// TIA Portal V16 export
// export: Created 2023-03-29T11:03:26.8705636Z, ExportSetting WithDefaults, DisplayName Totally Integrated Automation Portal, DisplayVersion V16 Update 6, DisplayName TIA Portal Version Control Interface, DisplayVersion V16 Update 2, DisplayName TIA Portal Openness, DisplayVersion V16 Update 6, DisplayName STEP 7 Professional, DisplayVersion V16 Update 6, DisplayName STEP 7 Safety, DisplayVersion V16, DisplayName WinCC Advanced, DisplayVersion V16 Update 6
FUNCTION "Read_MPP04_2_ModbusRTU" : Void   // FC24, LAD
TITLE = Odczyt parametrów z MPP04 Pompownia / Read data from SC100
{ S7_Optimized_Access := 'TRUE' }
AUTHOR : rtecmer
VERSION : 0.1
// Czytanie z przepływomierza pompownia główna. Modbus RTU 19200, bit stop-1, parti-no
// Czytanie z SC1000 
// Obsługa protokołu Master Modbus RTU.  Odczyt pomiarów  i status czujnika SC1000
// stored: AutoNumber false, IsIECCheckEnabled false, SetENOAutomatically false, UDAEnableTagReadback false
   VAR_TEMP
      Wielkość_przeływu_Adres0_0 : DWord;
      Wielkość_przeływu_Adres0_1 : DWord;
      Wielkość_przeływu_Adres2_0 : DWord;
      Wielkość_przeływu_Adres2_2 : DWord;
   END_VAR
   VAR_TEMP   // added for the SCL form of the ladder/FBD networks
      _w1 : Bool;
      _w2 : Bool;
   END_VAR
BEGIN

REGION Network 1: Odczyt parametrów z MPP04 Studnia na tłocznym
   // Czytanie z przepływomierza pompownia główna. Modbus RTU 19200, bit stop-1, parti-no
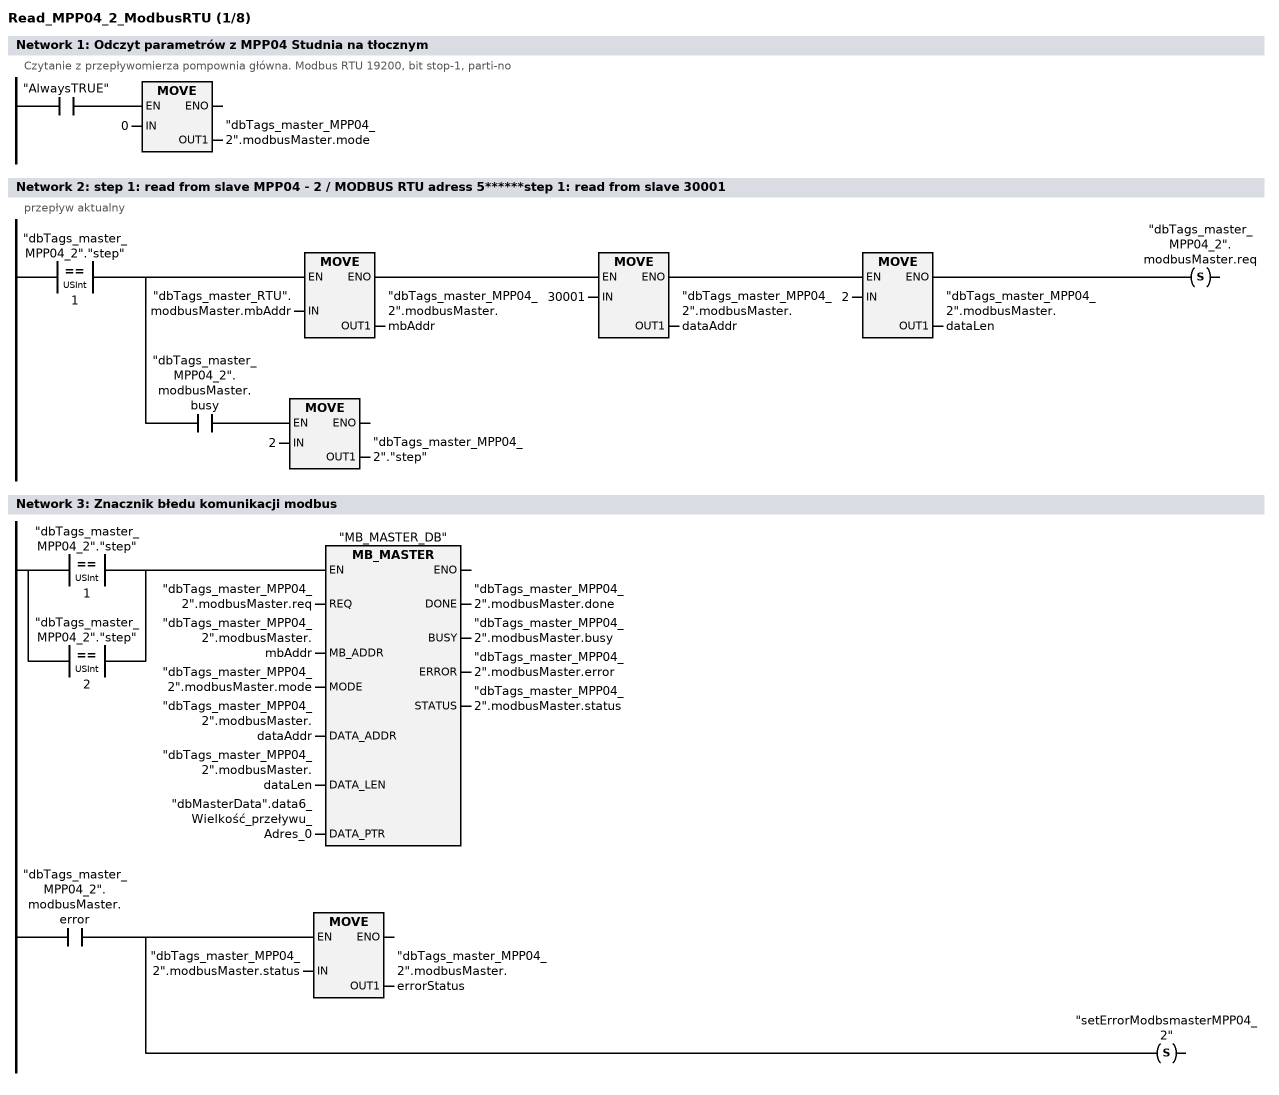
   RUNG wire#powerrail
      Contact( "AlwaysTRUE" )
      { S7_GenerateENO := "TRUE" } Move(in := 0, out1 => "dbTags_master_MPP04_2".modbusMaster.mode)
   END_RUNG
   // the same network as SCL:
   IF "AlwaysTRUE" THEN "dbTags_master_MPP04_2".modbusMaster.mode := 0; END_IF;
END_REGION

REGION Network 2: step 1: read from slave MPP04 - 2 / MODBUS RTU adress 5******step 1: read from slave 30001
   // przepływ aktualny
   RUNG wire#powerrail
      { S7_Templates := "SrcType := USInt" } EQ_Contact(in1 := "dbTags_master_MPP04_2"."step", in2 := 1)
      wire#w1
      Move(in := "dbTags_master_RTU".modbusMaster.mbAddr, out1 => "dbTags_master_MPP04_2".modbusMaster.mbAddr)
      { S7_GenerateENO := "TRUE" } Move(in := 30001, out1 => "dbTags_master_MPP04_2".modbusMaster.dataAddr)
      Move(in := 2, out1 => "dbTags_master_MPP04_2".modbusMaster.dataLen)
      S_Coil( "dbTags_master_MPP04_2".modbusMaster.req )
   END_RUNG
   RUNG wire#w1
      Contact( "dbTags_master_MPP04_2".modbusMaster.busy )
      { S7_GenerateENO := "TRUE" } Move(in := 2, out1 => "dbTags_master_MPP04_2"."step")
   END_RUNG
   // the same network as SCL:
   // ENO of a box is taken as its EN; it also drops when the box reports an error
   #_w1 := "dbTags_master_MPP04_2"."step" = 1;
   IF #_w1 THEN
       "dbTags_master_MPP04_2".modbusMaster.mbAddr := "dbTags_master_RTU".modbusMaster.mbAddr;
       "dbTags_master_MPP04_2".modbusMaster.dataAddr := 30001;
       "dbTags_master_MPP04_2".modbusMaster.dataLen := 2;
       "dbTags_master_MPP04_2".modbusMaster.req := TRUE;
   END_IF;
   IF #_w1 AND "dbTags_master_MPP04_2".modbusMaster.busy THEN "dbTags_master_MPP04_2"."step" := 2; END_IF;
END_REGION

REGION Network 3: Znacznik błedu komunikacji modbus
   RUNG wire#powerrail
      { S7_Templates := "SrcType := USInt" } EQ_Contact(in1 := "dbTags_master_MPP04_2"."step", in2 := 1)
      wire#w1
      "MB_MASTER_DB".MB_MASTER(REQ := "dbTags_master_MPP04_2".modbusMaster.req, MB_ADDR := "dbTags_master_MPP04_2".modbusMaster.mbAddr, MODE := "dbTags_master_MPP04_2".modbusMaster.mode, DATA_ADDR := "dbTags_master_MPP04_2".modbusMaster.dataAddr, DATA_LEN := "dbTags_master_MPP04_2".modbusMaster.dataLen, DATA_PTR := "dbMasterData".data6_Wielkość_przeływu_Adres_0, DONE => "dbTags_master_MPP04_2".modbusMaster.done, BUSY => "dbTags_master_MPP04_2".modbusMaster.busy, ERROR => "dbTags_master_MPP04_2".modbusMaster.error, STATUS => "dbTags_master_MPP04_2".modbusMaster.status)
   END_RUNG
   RUNG wire#powerrail
      { S7_Templates := "SrcType := USInt" } EQ_Contact(in1 := "dbTags_master_MPP04_2"."step", in2 := 2)
   END_RUNG wire#w1
   RUNG wire#powerrail
      Contact( "dbTags_master_MPP04_2".modbusMaster.error )
      wire#w2
      { S7_GenerateENO := "TRUE" } Move(in := "dbTags_master_MPP04_2".modbusMaster.status, out1 => "dbTags_master_MPP04_2".modbusMaster.errorStatus)
   END_RUNG
   RUNG wire#w2
      S_Coil( "setErrorModbsmasterMPP04_2" )
   END_RUNG
   // the same network as SCL:
   IF ("dbTags_master_MPP04_2"."step" = 1) OR ("dbTags_master_MPP04_2"."step" = 2) THEN
       "MB_MASTER_DB"(REQ := "dbTags_master_MPP04_2".modbusMaster.req,   // MB_MASTER
                      MB_ADDR := "dbTags_master_MPP04_2".modbusMaster.mbAddr,
                      MODE := "dbTags_master_MPP04_2".modbusMaster.mode,
                      DATA_ADDR := "dbTags_master_MPP04_2".modbusMaster.dataAddr,
                      DATA_LEN := "dbTags_master_MPP04_2".modbusMaster.dataLen,
                      DATA_PTR := "dbMasterData".data6_Wielkość_przeływu_Adres_0,
                      DONE => "dbTags_master_MPP04_2".modbusMaster.done,
                      BUSY => "dbTags_master_MPP04_2".modbusMaster.busy,
                      ERROR => "dbTags_master_MPP04_2".modbusMaster.error,
                      STATUS => "dbTags_master_MPP04_2".modbusMaster.status);
   END_IF;
   IF "dbTags_master_MPP04_2".modbusMaster.error THEN
       "dbTags_master_MPP04_2".modbusMaster.errorStatus := "dbTags_master_MPP04_2".modbusMaster.status;
       "setErrorModbsmasterMPP04_2" := TRUE;
   END_IF;
END_REGION

REGION Network 4: step 4: save received data / step 2: save received data 30001
   // Pomiar Temperatury KDN1
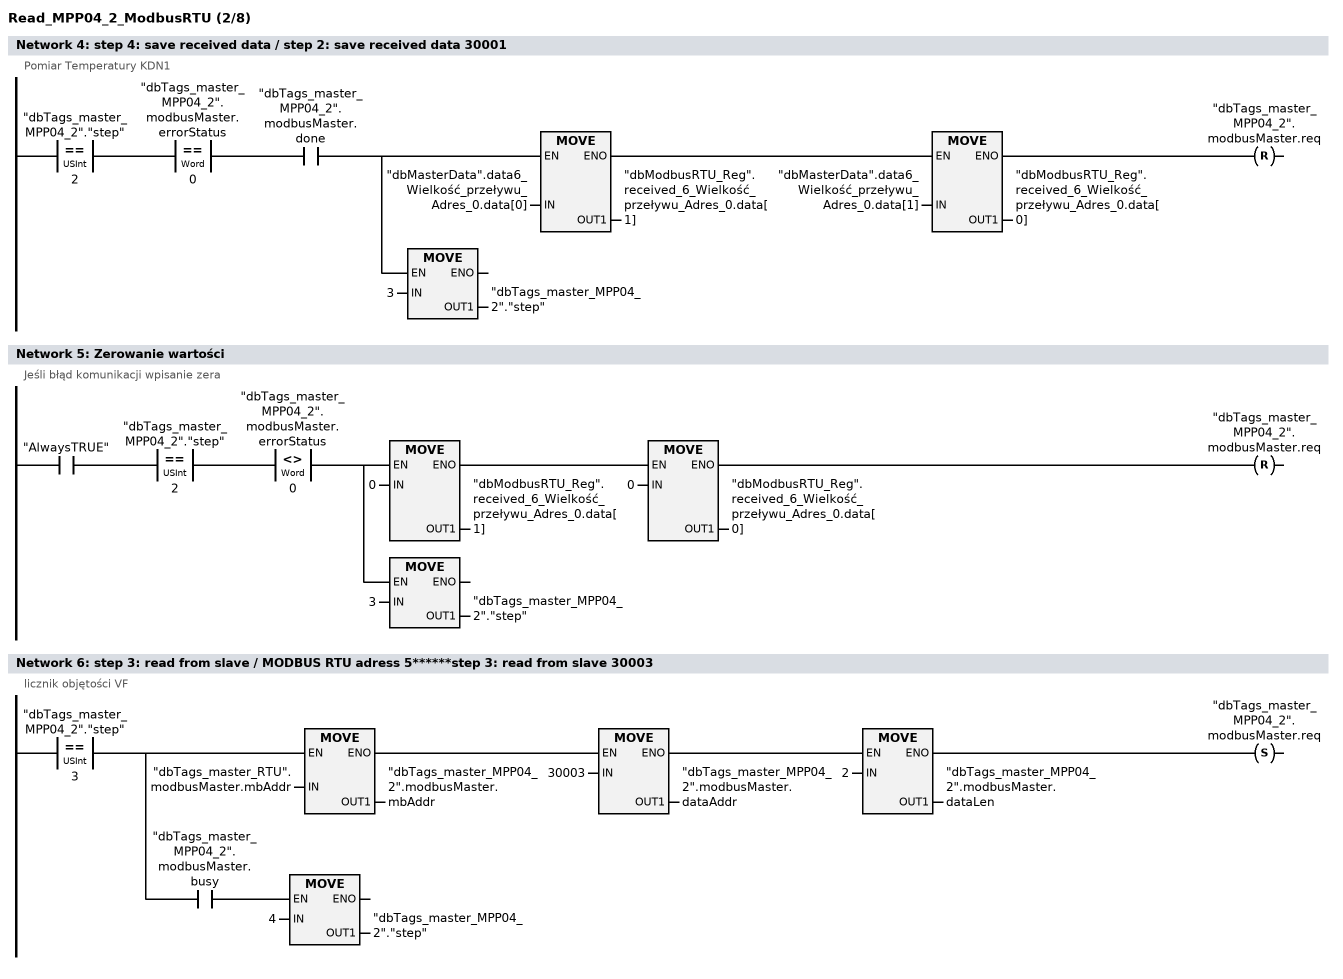
   RUNG wire#powerrail
      { S7_Templates := "SrcType := USInt" } EQ_Contact(in1 := "dbTags_master_MPP04_2"."step", in2 := 2)
      { S7_Templates := "SrcType := Word" } EQ_Contact(in1 := "dbTags_master_MPP04_2".modbusMaster.errorStatus, in2 := 0)
      Contact( "dbTags_master_MPP04_2".modbusMaster.done )
      wire#w1
      { S7_GenerateENO := "TRUE" } Move(in := "dbMasterData".data6_Wielkość_przeływu_Adres_0.data[0], out1 => "dbModbusRTU_Reg".received_6_Wielkość_przeływu_Adres_0.data[1])
      { S7_GenerateENO := "TRUE" } Move(in := "dbMasterData".data6_Wielkość_przeływu_Adres_0.data[1], out1 => "dbModbusRTU_Reg".received_6_Wielkość_przeływu_Adres_0.data[0])
      R_Coil( "dbTags_master_MPP04_2".modbusMaster.req )
   END_RUNG
   RUNG wire#w1
      { S7_GenerateENO := "TRUE" } Move(in := 3, out1 => "dbTags_master_MPP04_2"."step")
   END_RUNG
   // the same network as SCL:
   // ENO of a box is taken as its EN; it also drops when the box reports an error
   IF ("dbTags_master_MPP04_2"."step" = 2) AND ("dbTags_master_MPP04_2".modbusMaster.errorStatus = 0) AND "dbTags_master_MPP04_2".modbusMaster.done THEN
       "dbModbusRTU_Reg".received_6_Wielkość_przeływu_Adres_0.data[1] := "dbMasterData".data6_Wielkość_przeływu_Adres_0.data[0];
       "dbModbusRTU_Reg".received_6_Wielkość_przeływu_Adres_0.data[0] := "dbMasterData".data6_Wielkość_przeływu_Adres_0.data[1];
       "dbTags_master_MPP04_2".modbusMaster.req := FALSE;
       "dbTags_master_MPP04_2"."step" := 3;
   END_IF;
END_REGION

REGION Network 5: Zerowanie wartości
   // Jeśli błąd komunikacji wpisanie zera
   RUNG wire#powerrail
      Contact( "AlwaysTRUE" )
      { S7_Templates := "SrcType := USInt" } EQ_Contact(in1 := "dbTags_master_MPP04_2"."step", in2 := 2)
      { S7_Templates := "SrcType := Word" } NE_Contact(in1 := "dbTags_master_MPP04_2".modbusMaster.errorStatus, in2 := 0)
      wire#w1
      { S7_GenerateENO := "TRUE" } Move(in := 0, out1 => "dbModbusRTU_Reg".received_6_Wielkość_przeływu_Adres_0.data[1])
      { S7_GenerateENO := "TRUE" } Move(in := 0, out1 => "dbModbusRTU_Reg".received_6_Wielkość_przeływu_Adres_0.data[0])
      R_Coil( "dbTags_master_MPP04_2".modbusMaster.req )
   END_RUNG
   RUNG wire#w1
      { S7_GenerateENO := "TRUE" } Move(in := 3, out1 => "dbTags_master_MPP04_2"."step")
   END_RUNG
   // the same network as SCL:
   // ENO of a box is taken as its EN; it also drops when the box reports an error
   IF "AlwaysTRUE" AND ("dbTags_master_MPP04_2"."step" = 2) AND ("dbTags_master_MPP04_2".modbusMaster.errorStatus <> 0) THEN
       "dbModbusRTU_Reg".received_6_Wielkość_przeływu_Adres_0.data[1] := 0;
       "dbModbusRTU_Reg".received_6_Wielkość_przeływu_Adres_0.data[0] := 0;
       "dbTags_master_MPP04_2".modbusMaster.req := FALSE;
       "dbTags_master_MPP04_2"."step" := 3;
   END_IF;
END_REGION

REGION Network 6: step 3: read from slave / MODBUS RTU adress 5******step 3: read from slave 30003
   // licznik objętości VF
   RUNG wire#powerrail
      { S7_Templates := "SrcType := USInt" } EQ_Contact(in1 := "dbTags_master_MPP04_2"."step", in2 := 3)
      wire#w1
      Move(in := "dbTags_master_RTU".modbusMaster.mbAddr, out1 => "dbTags_master_MPP04_2".modbusMaster.mbAddr)
      { S7_GenerateENO := "TRUE" } Move(in := 30003, out1 => "dbTags_master_MPP04_2".modbusMaster.dataAddr)
      Move(in := 2, out1 => "dbTags_master_MPP04_2".modbusMaster.dataLen)
      S_Coil( "dbTags_master_MPP04_2".modbusMaster.req )
   END_RUNG
   RUNG wire#w1
      Contact( "dbTags_master_MPP04_2".modbusMaster.busy )
      { S7_GenerateENO := "TRUE" } Move(in := 4, out1 => "dbTags_master_MPP04_2"."step")
   END_RUNG
   // the same network as SCL:
   // ENO of a box is taken as its EN; it also drops when the box reports an error
   #_w1 := "dbTags_master_MPP04_2"."step" = 3;
   IF #_w1 THEN
       "dbTags_master_MPP04_2".modbusMaster.mbAddr := "dbTags_master_RTU".modbusMaster.mbAddr;
       "dbTags_master_MPP04_2".modbusMaster.dataAddr := 30003;
       "dbTags_master_MPP04_2".modbusMaster.dataLen := 2;
       "dbTags_master_MPP04_2".modbusMaster.req := TRUE;
   END_IF;
   IF #_w1 AND "dbTags_master_MPP04_2".modbusMaster.busy THEN "dbTags_master_MPP04_2"."step" := 4; END_IF;
END_REGION

REGION Network 7: Znacznik błedu komunikacji modbus
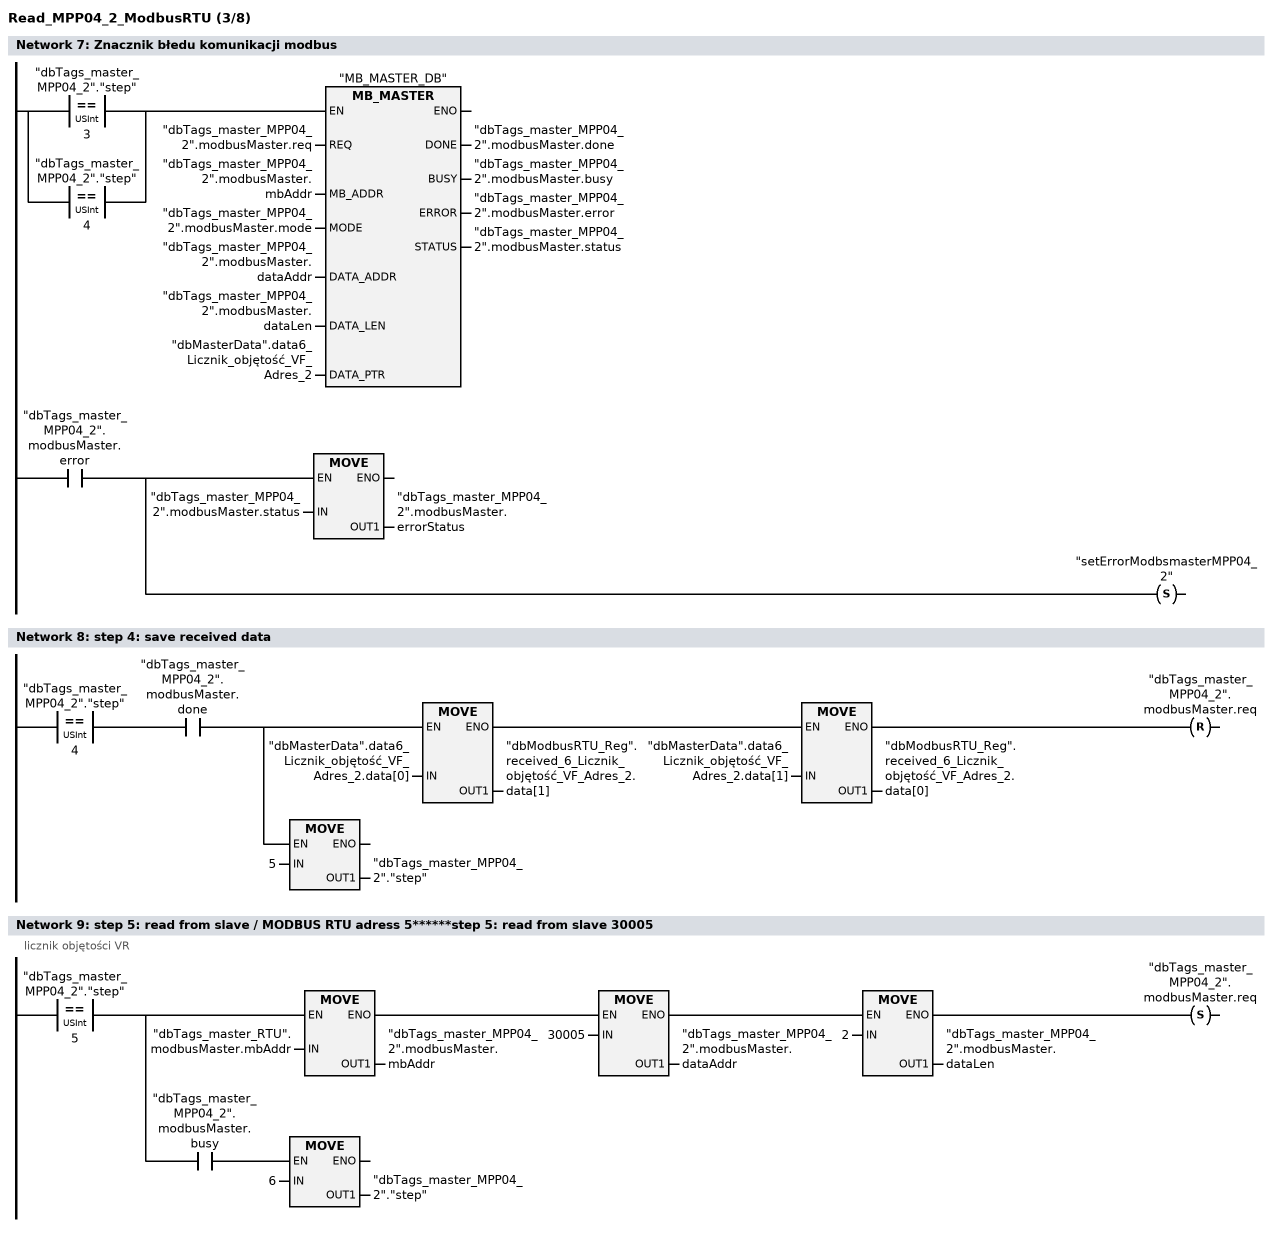
   RUNG wire#powerrail
      { S7_Templates := "SrcType := USInt" } EQ_Contact(in1 := "dbTags_master_MPP04_2"."step", in2 := 3)
      wire#w1
      "MB_MASTER_DB".MB_MASTER(REQ := "dbTags_master_MPP04_2".modbusMaster.req, MB_ADDR := "dbTags_master_MPP04_2".modbusMaster.mbAddr, MODE := "dbTags_master_MPP04_2".modbusMaster.mode, DATA_ADDR := "dbTags_master_MPP04_2".modbusMaster.dataAddr, DATA_LEN := "dbTags_master_MPP04_2".modbusMaster.dataLen, DATA_PTR := "dbMasterData".data6_Licznik_objętość_VF_Adres_2, DONE => "dbTags_master_MPP04_2".modbusMaster.done, BUSY => "dbTags_master_MPP04_2".modbusMaster.busy, ERROR => "dbTags_master_MPP04_2".modbusMaster.error, STATUS => "dbTags_master_MPP04_2".modbusMaster.status)
   END_RUNG
   RUNG wire#powerrail
      { S7_Templates := "SrcType := USInt" } EQ_Contact(in1 := "dbTags_master_MPP04_2"."step", in2 := 4)
   END_RUNG wire#w1
   RUNG wire#powerrail
      Contact( "dbTags_master_MPP04_2".modbusMaster.error )
      wire#w2
      { S7_GenerateENO := "TRUE" } Move(in := "dbTags_master_MPP04_2".modbusMaster.status, out1 => "dbTags_master_MPP04_2".modbusMaster.errorStatus)
   END_RUNG
   RUNG wire#w2
      S_Coil( "setErrorModbsmasterMPP04_2" )
   END_RUNG
   // the same network as SCL:
   IF ("dbTags_master_MPP04_2"."step" = 3) OR ("dbTags_master_MPP04_2"."step" = 4) THEN
       "MB_MASTER_DB"(REQ := "dbTags_master_MPP04_2".modbusMaster.req,   // MB_MASTER
                      MB_ADDR := "dbTags_master_MPP04_2".modbusMaster.mbAddr,
                      MODE := "dbTags_master_MPP04_2".modbusMaster.mode,
                      DATA_ADDR := "dbTags_master_MPP04_2".modbusMaster.dataAddr,
                      DATA_LEN := "dbTags_master_MPP04_2".modbusMaster.dataLen,
                      DATA_PTR := "dbMasterData".data6_Licznik_objętość_VF_Adres_2,
                      DONE => "dbTags_master_MPP04_2".modbusMaster.done,
                      BUSY => "dbTags_master_MPP04_2".modbusMaster.busy,
                      ERROR => "dbTags_master_MPP04_2".modbusMaster.error,
                      STATUS => "dbTags_master_MPP04_2".modbusMaster.status);
   END_IF;
   IF "dbTags_master_MPP04_2".modbusMaster.error THEN
       "dbTags_master_MPP04_2".modbusMaster.errorStatus := "dbTags_master_MPP04_2".modbusMaster.status;
       "setErrorModbsmasterMPP04_2" := TRUE;
   END_IF;
END_REGION

REGION Network 8: step 4: save received data
   RUNG wire#powerrail
      { S7_Templates := "SrcType := USInt" } EQ_Contact(in1 := "dbTags_master_MPP04_2"."step", in2 := 4)
      Contact( "dbTags_master_MPP04_2".modbusMaster.done )
      wire#w1
      { S7_GenerateENO := "TRUE" } Move(in := "dbMasterData".data6_Licznik_objętość_VF_Adres_2.data[0], out1 => "dbModbusRTU_Reg".received_6_Licznik_objętość_VF_Adres_2.data[1])
      { S7_GenerateENO := "TRUE" } Move(in := "dbMasterData".data6_Licznik_objętość_VF_Adres_2.data[1], out1 => "dbModbusRTU_Reg".received_6_Licznik_objętość_VF_Adres_2.data[0])
      R_Coil( "dbTags_master_MPP04_2".modbusMaster.req )
   END_RUNG
   RUNG wire#w1
      { S7_GenerateENO := "TRUE" } Move(in := 5, out1 => "dbTags_master_MPP04_2"."step")
   END_RUNG
   // the same network as SCL:
   // ENO of a box is taken as its EN; it also drops when the box reports an error
   IF ("dbTags_master_MPP04_2"."step" = 4) AND "dbTags_master_MPP04_2".modbusMaster.done THEN
       "dbModbusRTU_Reg".received_6_Licznik_objętość_VF_Adres_2.data[1] := "dbMasterData".data6_Licznik_objętość_VF_Adres_2.data[0];
       "dbModbusRTU_Reg".received_6_Licznik_objętość_VF_Adres_2.data[0] := "dbMasterData".data6_Licznik_objętość_VF_Adres_2.data[1];
       "dbTags_master_MPP04_2".modbusMaster.req := FALSE;
       "dbTags_master_MPP04_2"."step" := 5;
   END_IF;
END_REGION

REGION Network 9: step 5: read from slave / MODBUS RTU adress 5******step 5: read from slave 30005
   // licznik objętości VR
   RUNG wire#powerrail
      { S7_Templates := "SrcType := USInt" } EQ_Contact(in1 := "dbTags_master_MPP04_2"."step", in2 := 5)
      wire#w1
      Move(in := "dbTags_master_RTU".modbusMaster.mbAddr, out1 => "dbTags_master_MPP04_2".modbusMaster.mbAddr)
      { S7_GenerateENO := "TRUE" } Move(in := 30005, out1 => "dbTags_master_MPP04_2".modbusMaster.dataAddr)
      Move(in := 2, out1 => "dbTags_master_MPP04_2".modbusMaster.dataLen)
      S_Coil( "dbTags_master_MPP04_2".modbusMaster.req )
   END_RUNG
   RUNG wire#w1
      Contact( "dbTags_master_MPP04_2".modbusMaster.busy )
      { S7_GenerateENO := "TRUE" } Move(in := 6, out1 => "dbTags_master_MPP04_2"."step")
   END_RUNG
   // the same network as SCL:
   // ENO of a box is taken as its EN; it also drops when the box reports an error
   #_w1 := "dbTags_master_MPP04_2"."step" = 5;
   IF #_w1 THEN
       "dbTags_master_MPP04_2".modbusMaster.mbAddr := "dbTags_master_RTU".modbusMaster.mbAddr;
       "dbTags_master_MPP04_2".modbusMaster.dataAddr := 30005;
       "dbTags_master_MPP04_2".modbusMaster.dataLen := 2;
       "dbTags_master_MPP04_2".modbusMaster.req := TRUE;
   END_IF;
   IF #_w1 AND "dbTags_master_MPP04_2".modbusMaster.busy THEN "dbTags_master_MPP04_2"."step" := 6; END_IF;
END_REGION

REGION Network 10: Znacznik błedu komunikacji modbus
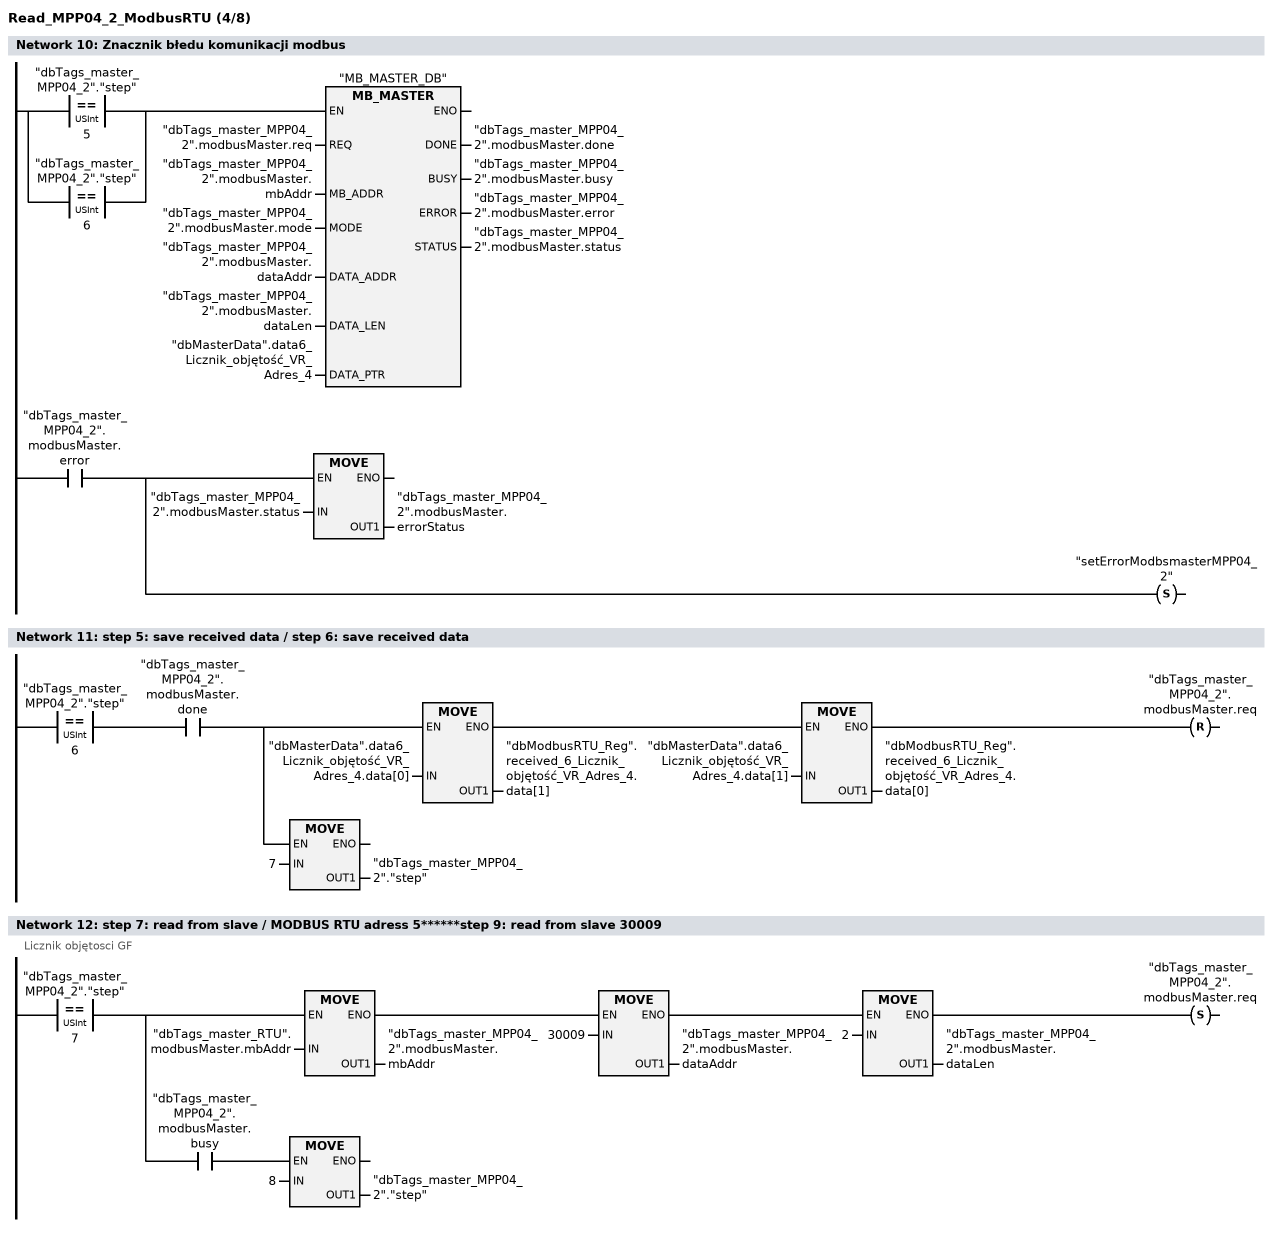
   RUNG wire#powerrail
      { S7_Templates := "SrcType := USInt" } EQ_Contact(in1 := "dbTags_master_MPP04_2"."step", in2 := 5)
      wire#w1
      "MB_MASTER_DB".MB_MASTER(REQ := "dbTags_master_MPP04_2".modbusMaster.req, MB_ADDR := "dbTags_master_MPP04_2".modbusMaster.mbAddr, MODE := "dbTags_master_MPP04_2".modbusMaster.mode, DATA_ADDR := "dbTags_master_MPP04_2".modbusMaster.dataAddr, DATA_LEN := "dbTags_master_MPP04_2".modbusMaster.dataLen, DATA_PTR := "dbMasterData".data6_Licznik_objętość_VR_Adres_4, DONE => "dbTags_master_MPP04_2".modbusMaster.done, BUSY => "dbTags_master_MPP04_2".modbusMaster.busy, ERROR => "dbTags_master_MPP04_2".modbusMaster.error, STATUS => "dbTags_master_MPP04_2".modbusMaster.status)
   END_RUNG
   RUNG wire#powerrail
      { S7_Templates := "SrcType := USInt" } EQ_Contact(in1 := "dbTags_master_MPP04_2"."step", in2 := 6)
   END_RUNG wire#w1
   RUNG wire#powerrail
      Contact( "dbTags_master_MPP04_2".modbusMaster.error )
      wire#w2
      { S7_GenerateENO := "TRUE" } Move(in := "dbTags_master_MPP04_2".modbusMaster.status, out1 => "dbTags_master_MPP04_2".modbusMaster.errorStatus)
   END_RUNG
   RUNG wire#w2
      S_Coil( "setErrorModbsmasterMPP04_2" )
   END_RUNG
   // the same network as SCL:
   IF ("dbTags_master_MPP04_2"."step" = 5) OR ("dbTags_master_MPP04_2"."step" = 6) THEN
       "MB_MASTER_DB"(REQ := "dbTags_master_MPP04_2".modbusMaster.req,   // MB_MASTER
                      MB_ADDR := "dbTags_master_MPP04_2".modbusMaster.mbAddr,
                      MODE := "dbTags_master_MPP04_2".modbusMaster.mode,
                      DATA_ADDR := "dbTags_master_MPP04_2".modbusMaster.dataAddr,
                      DATA_LEN := "dbTags_master_MPP04_2".modbusMaster.dataLen,
                      DATA_PTR := "dbMasterData".data6_Licznik_objętość_VR_Adres_4,
                      DONE => "dbTags_master_MPP04_2".modbusMaster.done,
                      BUSY => "dbTags_master_MPP04_2".modbusMaster.busy,
                      ERROR => "dbTags_master_MPP04_2".modbusMaster.error,
                      STATUS => "dbTags_master_MPP04_2".modbusMaster.status);
   END_IF;
   IF "dbTags_master_MPP04_2".modbusMaster.error THEN
       "dbTags_master_MPP04_2".modbusMaster.errorStatus := "dbTags_master_MPP04_2".modbusMaster.status;
       "setErrorModbsmasterMPP04_2" := TRUE;
   END_IF;
END_REGION

REGION Network 11: step 5: save received data / step 6: save received data
   RUNG wire#powerrail
      { S7_Templates := "SrcType := USInt" } EQ_Contact(in1 := "dbTags_master_MPP04_2"."step", in2 := 6)
      Contact( "dbTags_master_MPP04_2".modbusMaster.done )
      wire#w1
      { S7_GenerateENO := "TRUE" } Move(in := "dbMasterData".data6_Licznik_objętość_VR_Adres_4.data[0], out1 => "dbModbusRTU_Reg".received_6_Licznik_objętość_VR_Adres_4.data[1])
      { S7_GenerateENO := "TRUE" } Move(in := "dbMasterData".data6_Licznik_objętość_VR_Adres_4.data[1], out1 => "dbModbusRTU_Reg".received_6_Licznik_objętość_VR_Adres_4.data[0])
      R_Coil( "dbTags_master_MPP04_2".modbusMaster.req )
   END_RUNG
   RUNG wire#w1
      { S7_GenerateENO := "TRUE" } Move(in := 7, out1 => "dbTags_master_MPP04_2"."step")
   END_RUNG
   // the same network as SCL:
   // ENO of a box is taken as its EN; it also drops when the box reports an error
   IF ("dbTags_master_MPP04_2"."step" = 6) AND "dbTags_master_MPP04_2".modbusMaster.done THEN
       "dbModbusRTU_Reg".received_6_Licznik_objętość_VR_Adres_4.data[1] := "dbMasterData".data6_Licznik_objętość_VR_Adres_4.data[0];
       "dbModbusRTU_Reg".received_6_Licznik_objętość_VR_Adres_4.data[0] := "dbMasterData".data6_Licznik_objętość_VR_Adres_4.data[1];
       "dbTags_master_MPP04_2".modbusMaster.req := FALSE;
       "dbTags_master_MPP04_2"."step" := 7;
   END_IF;
END_REGION

REGION Network 12: step 7: read from slave / MODBUS RTU adress 5******step 9: read from slave 30009
   // Licznik objętosci GF
   RUNG wire#powerrail
      { S7_Templates := "SrcType := USInt" } EQ_Contact(in1 := "dbTags_master_MPP04_2"."step", in2 := 7)
      wire#w1
      Move(in := "dbTags_master_RTU".modbusMaster.mbAddr, out1 => "dbTags_master_MPP04_2".modbusMaster.mbAddr)
      { S7_GenerateENO := "TRUE" } Move(in := 30009, out1 => "dbTags_master_MPP04_2".modbusMaster.dataAddr)
      Move(in := 2, out1 => "dbTags_master_MPP04_2".modbusMaster.dataLen)
      S_Coil( "dbTags_master_MPP04_2".modbusMaster.req )
   END_RUNG
   RUNG wire#w1
      Contact( "dbTags_master_MPP04_2".modbusMaster.busy )
      { S7_GenerateENO := "TRUE" } Move(in := 8, out1 => "dbTags_master_MPP04_2"."step")
   END_RUNG
   // the same network as SCL:
   // ENO of a box is taken as its EN; it also drops when the box reports an error
   #_w1 := "dbTags_master_MPP04_2"."step" = 7;
   IF #_w1 THEN
       "dbTags_master_MPP04_2".modbusMaster.mbAddr := "dbTags_master_RTU".modbusMaster.mbAddr;
       "dbTags_master_MPP04_2".modbusMaster.dataAddr := 30009;
       "dbTags_master_MPP04_2".modbusMaster.dataLen := 2;
       "dbTags_master_MPP04_2".modbusMaster.req := TRUE;
   END_IF;
   IF #_w1 AND "dbTags_master_MPP04_2".modbusMaster.busy THEN "dbTags_master_MPP04_2"."step" := 8; END_IF;
END_REGION

REGION Network 13: Znacznik błedu komunikacji modbus
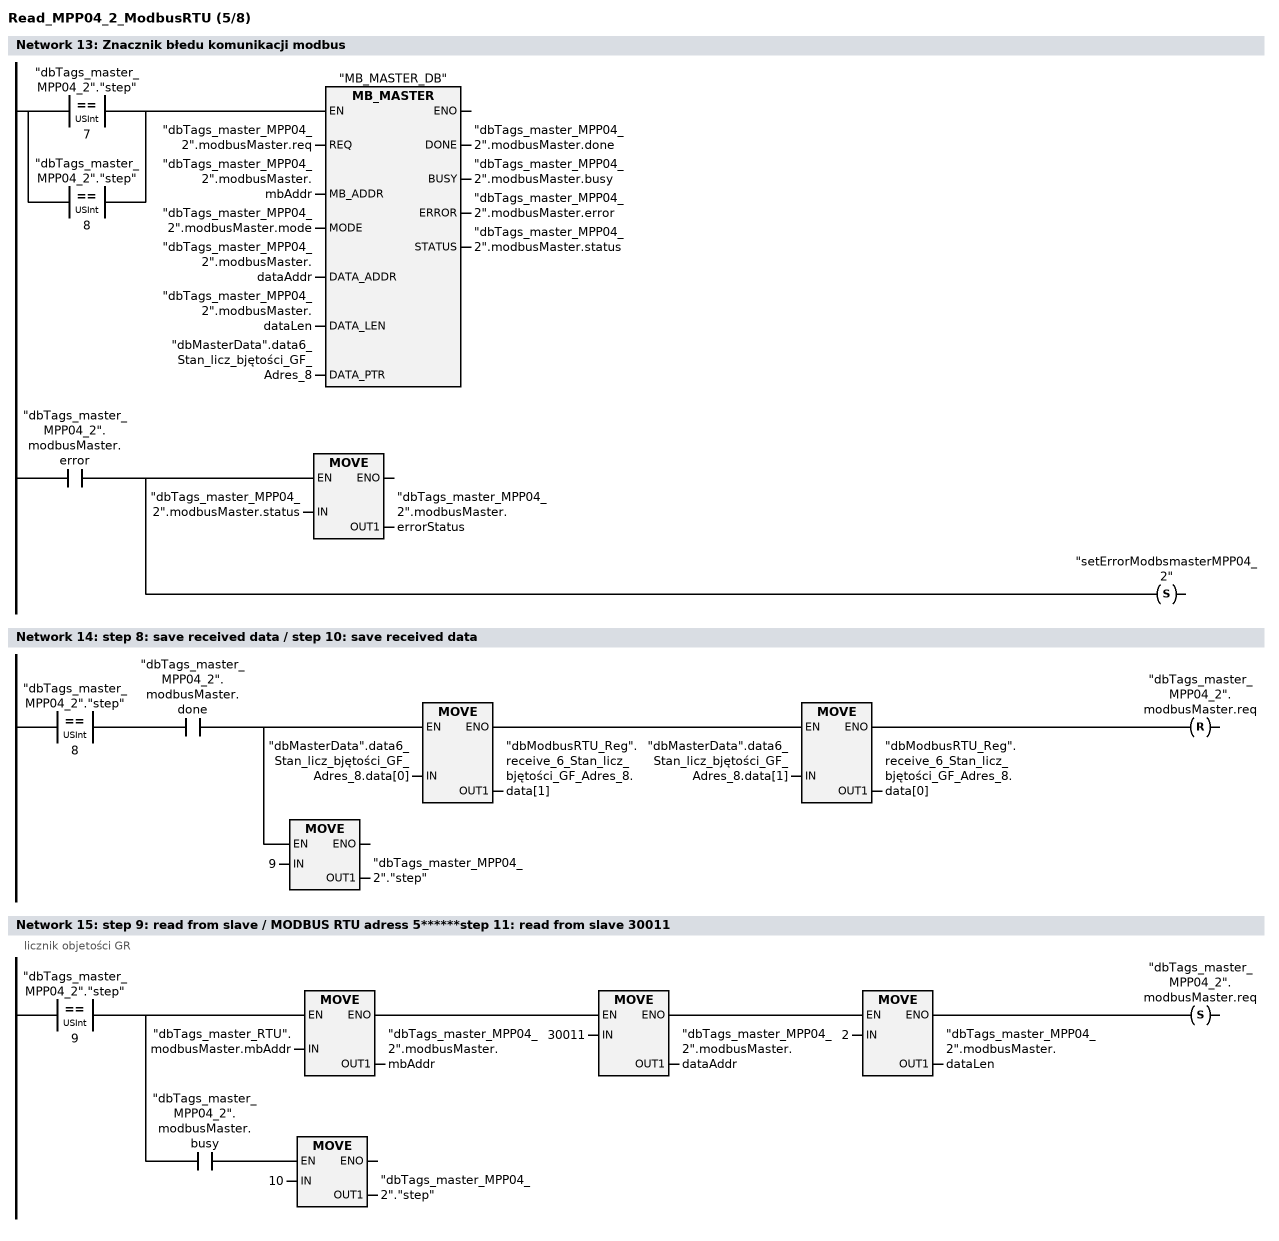
   RUNG wire#powerrail
      { S7_Templates := "SrcType := USInt" } EQ_Contact(in1 := "dbTags_master_MPP04_2"."step", in2 := 7)
      wire#w1
      "MB_MASTER_DB".MB_MASTER(REQ := "dbTags_master_MPP04_2".modbusMaster.req, MB_ADDR := "dbTags_master_MPP04_2".modbusMaster.mbAddr, MODE := "dbTags_master_MPP04_2".modbusMaster.mode, DATA_ADDR := "dbTags_master_MPP04_2".modbusMaster.dataAddr, DATA_LEN := "dbTags_master_MPP04_2".modbusMaster.dataLen, DATA_PTR := "dbMasterData".data6_Stan_licz_bjętości_GF_Adres_8, DONE => "dbTags_master_MPP04_2".modbusMaster.done, BUSY => "dbTags_master_MPP04_2".modbusMaster.busy, ERROR => "dbTags_master_MPP04_2".modbusMaster.error, STATUS => "dbTags_master_MPP04_2".modbusMaster.status)
   END_RUNG
   RUNG wire#powerrail
      { S7_Templates := "SrcType := USInt" } EQ_Contact(in1 := "dbTags_master_MPP04_2"."step", in2 := 8)
   END_RUNG wire#w1
   RUNG wire#powerrail
      Contact( "dbTags_master_MPP04_2".modbusMaster.error )
      wire#w2
      { S7_GenerateENO := "TRUE" } Move(in := "dbTags_master_MPP04_2".modbusMaster.status, out1 => "dbTags_master_MPP04_2".modbusMaster.errorStatus)
   END_RUNG
   RUNG wire#w2
      S_Coil( "setErrorModbsmasterMPP04_2" )
   END_RUNG
   // the same network as SCL:
   IF ("dbTags_master_MPP04_2"."step" = 7) OR ("dbTags_master_MPP04_2"."step" = 8) THEN
       "MB_MASTER_DB"(REQ := "dbTags_master_MPP04_2".modbusMaster.req,   // MB_MASTER
                      MB_ADDR := "dbTags_master_MPP04_2".modbusMaster.mbAddr,
                      MODE := "dbTags_master_MPP04_2".modbusMaster.mode,
                      DATA_ADDR := "dbTags_master_MPP04_2".modbusMaster.dataAddr,
                      DATA_LEN := "dbTags_master_MPP04_2".modbusMaster.dataLen,
                      DATA_PTR := "dbMasterData".data6_Stan_licz_bjętości_GF_Adres_8,
                      DONE => "dbTags_master_MPP04_2".modbusMaster.done,
                      BUSY => "dbTags_master_MPP04_2".modbusMaster.busy,
                      ERROR => "dbTags_master_MPP04_2".modbusMaster.error,
                      STATUS => "dbTags_master_MPP04_2".modbusMaster.status);
   END_IF;
   IF "dbTags_master_MPP04_2".modbusMaster.error THEN
       "dbTags_master_MPP04_2".modbusMaster.errorStatus := "dbTags_master_MPP04_2".modbusMaster.status;
       "setErrorModbsmasterMPP04_2" := TRUE;
   END_IF;
END_REGION

REGION Network 14: step 8: save received data / step 10: save received data
   RUNG wire#powerrail
      { S7_Templates := "SrcType := USInt" } EQ_Contact(in1 := "dbTags_master_MPP04_2"."step", in2 := 8)
      Contact( "dbTags_master_MPP04_2".modbusMaster.done )
      wire#w1
      { S7_GenerateENO := "TRUE" } Move(in := "dbMasterData".data6_Stan_licz_bjętości_GF_Adres_8.data[0], out1 => "dbModbusRTU_Reg".receive_6_Stan_licz_bjętości_GF_Adres_8.data[1])
      { S7_GenerateENO := "TRUE" } Move(in := "dbMasterData".data6_Stan_licz_bjętości_GF_Adres_8.data[1], out1 => "dbModbusRTU_Reg".receive_6_Stan_licz_bjętości_GF_Adres_8.data[0])
      R_Coil( "dbTags_master_MPP04_2".modbusMaster.req )
   END_RUNG
   RUNG wire#w1
      { S7_GenerateENO := "TRUE" } Move(in := 9, out1 => "dbTags_master_MPP04_2"."step")
   END_RUNG
   // the same network as SCL:
   // ENO of a box is taken as its EN; it also drops when the box reports an error
   IF ("dbTags_master_MPP04_2"."step" = 8) AND "dbTags_master_MPP04_2".modbusMaster.done THEN
       "dbModbusRTU_Reg".receive_6_Stan_licz_bjętości_GF_Adres_8.data[1] := "dbMasterData".data6_Stan_licz_bjętości_GF_Adres_8.data[0];
       "dbModbusRTU_Reg".receive_6_Stan_licz_bjętości_GF_Adres_8.data[0] := "dbMasterData".data6_Stan_licz_bjętości_GF_Adres_8.data[1];
       "dbTags_master_MPP04_2".modbusMaster.req := FALSE;
       "dbTags_master_MPP04_2"."step" := 9;
   END_IF;
END_REGION

REGION Network 15: step 9: read from slave / MODBUS RTU adress 5******step 11: read from slave 30011
   // licznik objetości GR
   RUNG wire#powerrail
      { S7_Templates := "SrcType := USInt" } EQ_Contact(in1 := "dbTags_master_MPP04_2"."step", in2 := 9)
      wire#w1
      Move(in := "dbTags_master_RTU".modbusMaster.mbAddr, out1 => "dbTags_master_MPP04_2".modbusMaster.mbAddr)
      { S7_GenerateENO := "TRUE" } Move(in := 30011, out1 => "dbTags_master_MPP04_2".modbusMaster.dataAddr)
      Move(in := 2, out1 => "dbTags_master_MPP04_2".modbusMaster.dataLen)
      S_Coil( "dbTags_master_MPP04_2".modbusMaster.req )
   END_RUNG
   RUNG wire#w1
      Contact( "dbTags_master_MPP04_2".modbusMaster.busy )
      { S7_GenerateENO := "TRUE" } Move(in := 10, out1 => "dbTags_master_MPP04_2"."step")
   END_RUNG
   // the same network as SCL:
   // ENO of a box is taken as its EN; it also drops when the box reports an error
   #_w1 := "dbTags_master_MPP04_2"."step" = 9;
   IF #_w1 THEN
       "dbTags_master_MPP04_2".modbusMaster.mbAddr := "dbTags_master_RTU".modbusMaster.mbAddr;
       "dbTags_master_MPP04_2".modbusMaster.dataAddr := 30011;
       "dbTags_master_MPP04_2".modbusMaster.dataLen := 2;
       "dbTags_master_MPP04_2".modbusMaster.req := TRUE;
   END_IF;
   IF #_w1 AND "dbTags_master_MPP04_2".modbusMaster.busy THEN "dbTags_master_MPP04_2"."step" := 10; END_IF;
END_REGION

REGION Network 16: Znacznik błedu komunikacji modbus
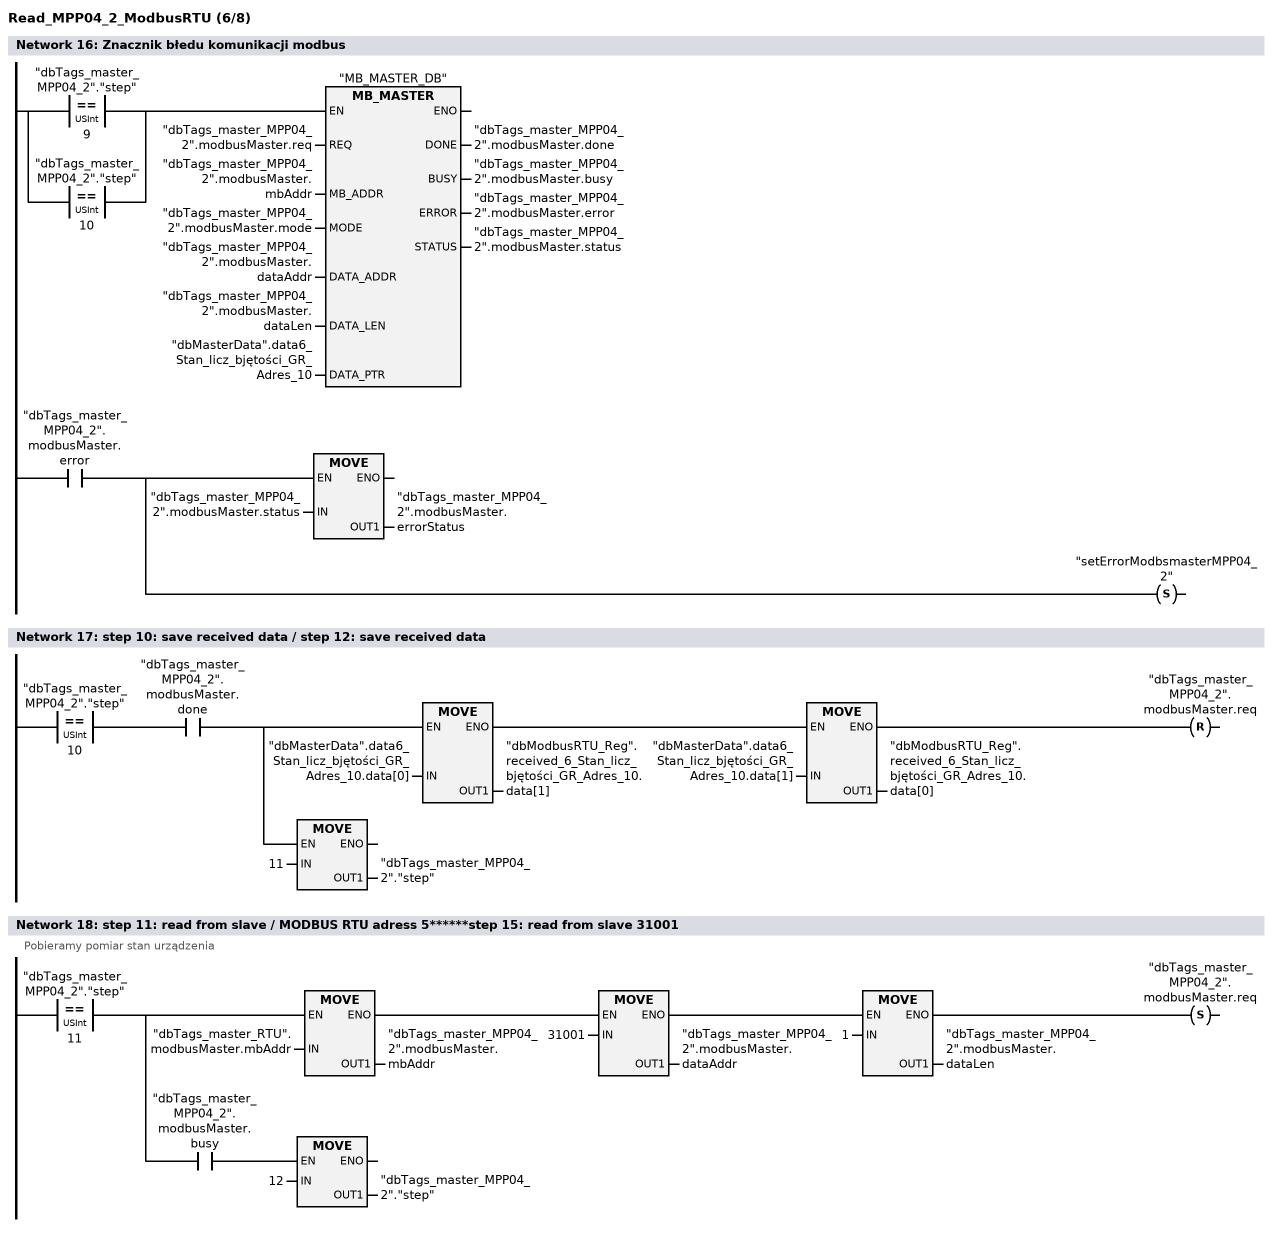
   RUNG wire#powerrail
      { S7_Templates := "SrcType := USInt" } EQ_Contact(in1 := "dbTags_master_MPP04_2"."step", in2 := 9)
      wire#w1
      "MB_MASTER_DB".MB_MASTER(REQ := "dbTags_master_MPP04_2".modbusMaster.req, MB_ADDR := "dbTags_master_MPP04_2".modbusMaster.mbAddr, MODE := "dbTags_master_MPP04_2".modbusMaster.mode, DATA_ADDR := "dbTags_master_MPP04_2".modbusMaster.dataAddr, DATA_LEN := "dbTags_master_MPP04_2".modbusMaster.dataLen, DATA_PTR := "dbMasterData".data6_Stan_licz_bjętości_GR_Adres_10, DONE => "dbTags_master_MPP04_2".modbusMaster.done, BUSY => "dbTags_master_MPP04_2".modbusMaster.busy, ERROR => "dbTags_master_MPP04_2".modbusMaster.error, STATUS => "dbTags_master_MPP04_2".modbusMaster.status)
   END_RUNG
   RUNG wire#powerrail
      { S7_Templates := "SrcType := USInt" } EQ_Contact(in1 := "dbTags_master_MPP04_2"."step", in2 := 10)
   END_RUNG wire#w1
   RUNG wire#powerrail
      Contact( "dbTags_master_MPP04_2".modbusMaster.error )
      wire#w2
      { S7_GenerateENO := "TRUE" } Move(in := "dbTags_master_MPP04_2".modbusMaster.status, out1 => "dbTags_master_MPP04_2".modbusMaster.errorStatus)
   END_RUNG
   RUNG wire#w2
      S_Coil( "setErrorModbsmasterMPP04_2" )
   END_RUNG
   // the same network as SCL:
   IF ("dbTags_master_MPP04_2"."step" = 9) OR ("dbTags_master_MPP04_2"."step" = 10) THEN
       "MB_MASTER_DB"(REQ := "dbTags_master_MPP04_2".modbusMaster.req,   // MB_MASTER
                      MB_ADDR := "dbTags_master_MPP04_2".modbusMaster.mbAddr,
                      MODE := "dbTags_master_MPP04_2".modbusMaster.mode,
                      DATA_ADDR := "dbTags_master_MPP04_2".modbusMaster.dataAddr,
                      DATA_LEN := "dbTags_master_MPP04_2".modbusMaster.dataLen,
                      DATA_PTR := "dbMasterData".data6_Stan_licz_bjętości_GR_Adres_10,
                      DONE => "dbTags_master_MPP04_2".modbusMaster.done,
                      BUSY => "dbTags_master_MPP04_2".modbusMaster.busy,
                      ERROR => "dbTags_master_MPP04_2".modbusMaster.error,
                      STATUS => "dbTags_master_MPP04_2".modbusMaster.status);
   END_IF;
   IF "dbTags_master_MPP04_2".modbusMaster.error THEN
       "dbTags_master_MPP04_2".modbusMaster.errorStatus := "dbTags_master_MPP04_2".modbusMaster.status;
       "setErrorModbsmasterMPP04_2" := TRUE;
   END_IF;
END_REGION

REGION Network 17: step 10: save received data / step 12: save received data
   RUNG wire#powerrail
      { S7_Templates := "SrcType := USInt" } EQ_Contact(in1 := "dbTags_master_MPP04_2"."step", in2 := 10)
      Contact( "dbTags_master_MPP04_2".modbusMaster.done )
      wire#w1
      { S7_GenerateENO := "TRUE" } Move(in := "dbMasterData".data6_Stan_licz_bjętości_GR_Adres_10.data[0], out1 => "dbModbusRTU_Reg".received_6_Stan_licz_bjętości_GR_Adres_10.data[1])
      { S7_GenerateENO := "TRUE" } Move(in := "dbMasterData".data6_Stan_licz_bjętości_GR_Adres_10.data[1], out1 => "dbModbusRTU_Reg".received_6_Stan_licz_bjętości_GR_Adres_10.data[0])
      R_Coil( "dbTags_master_MPP04_2".modbusMaster.req )
   END_RUNG
   RUNG wire#w1
      { S7_GenerateENO := "TRUE" } Move(in := 11, out1 => "dbTags_master_MPP04_2"."step")
   END_RUNG
   // the same network as SCL:
   // ENO of a box is taken as its EN; it also drops when the box reports an error
   IF ("dbTags_master_MPP04_2"."step" = 10) AND "dbTags_master_MPP04_2".modbusMaster.done THEN
       "dbModbusRTU_Reg".received_6_Stan_licz_bjętości_GR_Adres_10.data[1] := "dbMasterData".data6_Stan_licz_bjętości_GR_Adres_10.data[0];
       "dbModbusRTU_Reg".received_6_Stan_licz_bjętości_GR_Adres_10.data[0] := "dbMasterData".data6_Stan_licz_bjętości_GR_Adres_10.data[1];
       "dbTags_master_MPP04_2".modbusMaster.req := FALSE;
       "dbTags_master_MPP04_2"."step" := 11;
   END_IF;
END_REGION

REGION Network 18: step 11: read from slave / MODBUS RTU adress 5******step 15: read from slave 31001
   // Pobieramy pomiar stan urządzenia
   RUNG wire#powerrail
      { S7_Templates := "SrcType := USInt" } EQ_Contact(in1 := "dbTags_master_MPP04_2"."step", in2 := 11)
      wire#w1
      Move(in := "dbTags_master_RTU".modbusMaster.mbAddr, out1 => "dbTags_master_MPP04_2".modbusMaster.mbAddr)
      { S7_GenerateENO := "TRUE" } Move(in := 31001, out1 => "dbTags_master_MPP04_2".modbusMaster.dataAddr)
      Move(in := 1, out1 => "dbTags_master_MPP04_2".modbusMaster.dataLen)
      S_Coil( "dbTags_master_MPP04_2".modbusMaster.req )
   END_RUNG
   RUNG wire#w1
      Contact( "dbTags_master_MPP04_2".modbusMaster.busy )
      { S7_GenerateENO := "TRUE" } Move(in := 12, out1 => "dbTags_master_MPP04_2"."step")
   END_RUNG
   // the same network as SCL:
   // ENO of a box is taken as its EN; it also drops when the box reports an error
   #_w1 := "dbTags_master_MPP04_2"."step" = 11;
   IF #_w1 THEN
       "dbTags_master_MPP04_2".modbusMaster.mbAddr := "dbTags_master_RTU".modbusMaster.mbAddr;
       "dbTags_master_MPP04_2".modbusMaster.dataAddr := 31001;
       "dbTags_master_MPP04_2".modbusMaster.dataLen := 1;
       "dbTags_master_MPP04_2".modbusMaster.req := TRUE;
   END_IF;
   IF #_w1 AND "dbTags_master_MPP04_2".modbusMaster.busy THEN "dbTags_master_MPP04_2"."step" := 12; END_IF;
END_REGION

REGION Network 19: Znacznik błedu komunikacji modbus
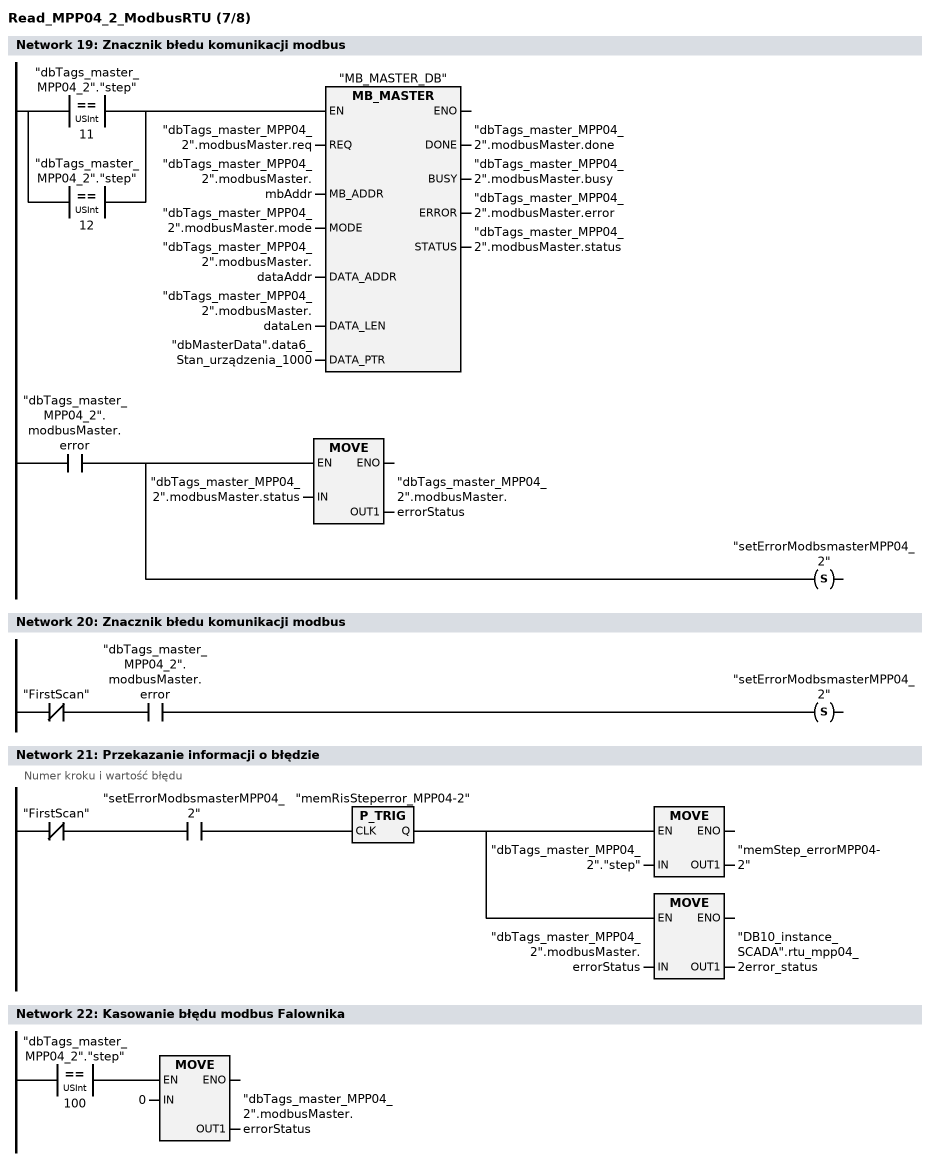
   RUNG wire#powerrail
      { S7_Templates := "SrcType := USInt" } EQ_Contact(in1 := "dbTags_master_MPP04_2"."step", in2 := 11)
      wire#w1
      "MB_MASTER_DB".MB_MASTER(REQ := "dbTags_master_MPP04_2".modbusMaster.req, MB_ADDR := "dbTags_master_MPP04_2".modbusMaster.mbAddr, MODE := "dbTags_master_MPP04_2".modbusMaster.mode, DATA_ADDR := "dbTags_master_MPP04_2".modbusMaster.dataAddr, DATA_LEN := "dbTags_master_MPP04_2".modbusMaster.dataLen, DATA_PTR := "dbMasterData".data6_Stan_urządzenia_1000, DONE => "dbTags_master_MPP04_2".modbusMaster.done, BUSY => "dbTags_master_MPP04_2".modbusMaster.busy, ERROR => "dbTags_master_MPP04_2".modbusMaster.error, STATUS => "dbTags_master_MPP04_2".modbusMaster.status)
   END_RUNG
   RUNG wire#powerrail
      { S7_Templates := "SrcType := USInt" } EQ_Contact(in1 := "dbTags_master_MPP04_2"."step", in2 := 12)
   END_RUNG wire#w1
   RUNG wire#powerrail
      Contact( "dbTags_master_MPP04_2".modbusMaster.error )
      wire#w2
      { S7_GenerateENO := "TRUE" } Move(in := "dbTags_master_MPP04_2".modbusMaster.status, out1 => "dbTags_master_MPP04_2".modbusMaster.errorStatus)
   END_RUNG
   RUNG wire#w2
      S_Coil( "setErrorModbsmasterMPP04_2" )
   END_RUNG
   // the same network as SCL:
   IF ("dbTags_master_MPP04_2"."step" = 11) OR ("dbTags_master_MPP04_2"."step" = 12) THEN
       "MB_MASTER_DB"(REQ := "dbTags_master_MPP04_2".modbusMaster.req,   // MB_MASTER
                      MB_ADDR := "dbTags_master_MPP04_2".modbusMaster.mbAddr,
                      MODE := "dbTags_master_MPP04_2".modbusMaster.mode,
                      DATA_ADDR := "dbTags_master_MPP04_2".modbusMaster.dataAddr,
                      DATA_LEN := "dbTags_master_MPP04_2".modbusMaster.dataLen,
                      DATA_PTR := "dbMasterData".data6_Stan_urządzenia_1000,
                      DONE => "dbTags_master_MPP04_2".modbusMaster.done,
                      BUSY => "dbTags_master_MPP04_2".modbusMaster.busy,
                      ERROR => "dbTags_master_MPP04_2".modbusMaster.error,
                      STATUS => "dbTags_master_MPP04_2".modbusMaster.status);
   END_IF;
   IF "dbTags_master_MPP04_2".modbusMaster.error THEN
       "dbTags_master_MPP04_2".modbusMaster.errorStatus := "dbTags_master_MPP04_2".modbusMaster.status;
       "setErrorModbsmasterMPP04_2" := TRUE;
   END_IF;
END_REGION

REGION Network 20: Znacznik błedu komunikacji modbus
   RUNG wire#powerrail
      I_Contact( "FirstScan" )
      Contact( "dbTags_master_MPP04_2".modbusMaster.error )
      S_Coil( "setErrorModbsmasterMPP04_2" )
   END_RUNG
   // the same network as SCL:
   IF NOT "FirstScan" AND "dbTags_master_MPP04_2".modbusMaster.error THEN
       "setErrorModbsmasterMPP04_2" := TRUE;
   END_IF;
END_REGION

REGION Network 21: Przekazanie informacji o błędzie
   // Numer kroku i wartość błędu
   RUNG wire#powerrail
      I_Contact( "FirstScan" )
      Contact( "setErrorModbsmasterMPP04_2" )
      P_Trig( "memRisSteperror_MPP04-2" )
      wire#w1
      Move(in := "dbTags_master_MPP04_2"."step", out1 => "memStep_errorMPP04-2")
   END_RUNG
   RUNG wire#w1
      { S7_GenerateENO := "TRUE" } Move(in := "dbTags_master_MPP04_2".modbusMaster.errorStatus, out1 => "DB10_instance_SCADA".rtu_mpp04_2error_status)
   END_RUNG
   // the same network as SCL:
   #_w1 := NOT "FirstScan" AND "setErrorModbsmasterMPP04_2";
   #_w2 := #_w1 AND NOT "memRisSteperror_MPP04-2";   // rising edge
   "memRisSteperror_MPP04-2" := #_w1;
   IF #_w2 THEN
       "memStep_errorMPP04-2" := "dbTags_master_MPP04_2"."step";
       "DB10_instance_SCADA".rtu_mpp04_2error_status := "dbTags_master_MPP04_2".modbusMaster.errorStatus;
   END_IF;
END_REGION

REGION Network 22: Kasowanie błędu modbus Falownika
   RUNG wire#powerrail
      { S7_Templates := "SrcType := USInt" } EQ_Contact(in1 := "dbTags_master_MPP04_2"."step", in2 := 100)
      { S7_GenerateENO := "TRUE" } Move(in := 0, out1 => "dbTags_master_MPP04_2".modbusMaster.errorStatus)
   END_RUNG
   // the same network as SCL:
   IF "dbTags_master_MPP04_2"."step" = 100 THEN
       "dbTags_master_MPP04_2".modbusMaster.errorStatus := 0;
   END_IF;
END_REGION

REGION Network 23: The enable to initiate a Modbus master request / step 16: save received data
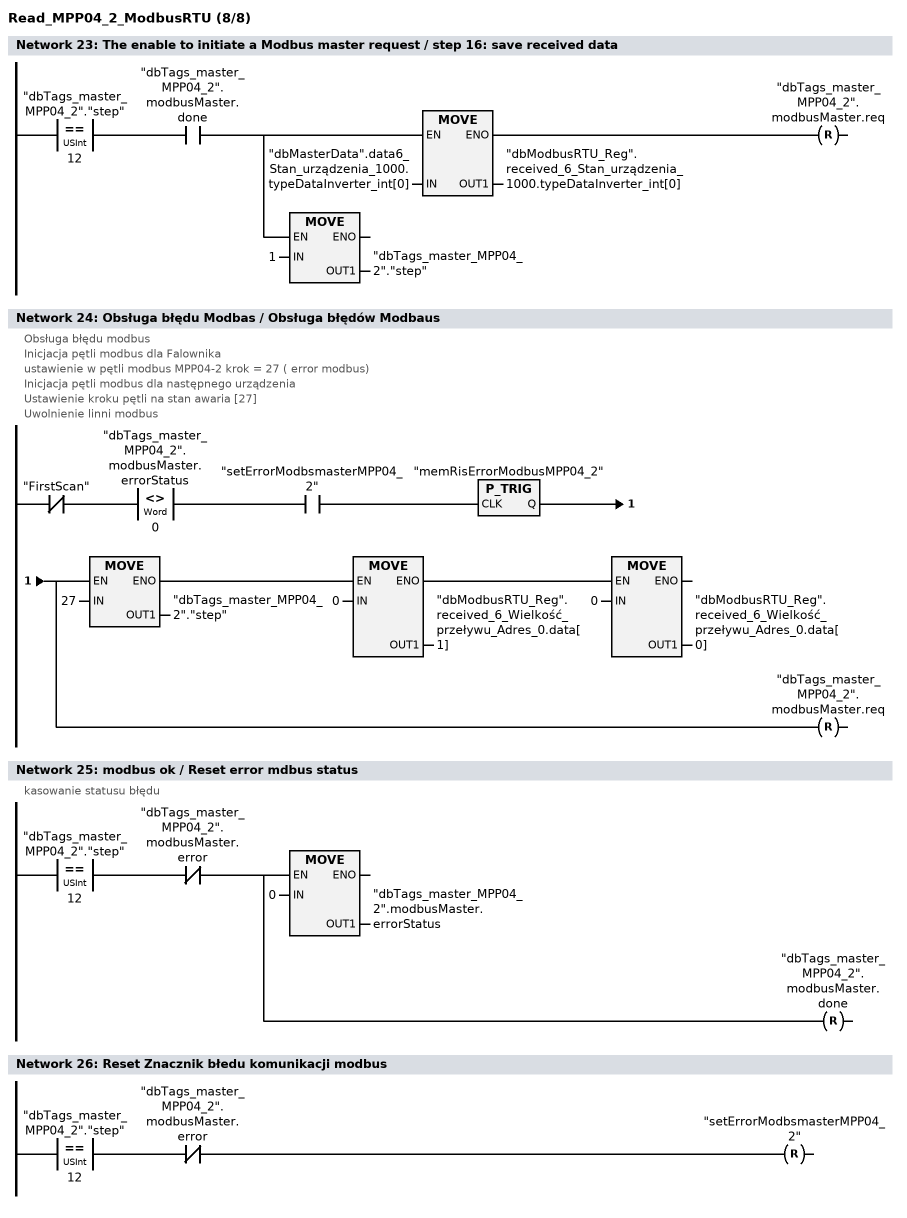
   RUNG wire#powerrail
      { S7_Templates := "SrcType := USInt" } EQ_Contact(in1 := "dbTags_master_MPP04_2"."step", in2 := 12)
      Contact( "dbTags_master_MPP04_2".modbusMaster.done )
      wire#w1
      { S7_GenerateENO := "TRUE" } Move(in := "dbMasterData".data6_Stan_urządzenia_1000.typeDataInverter_int[0], out1 => "dbModbusRTU_Reg".received_6_Stan_urządzenia_1000.typeDataInverter_int[0])
      R_Coil( "dbTags_master_MPP04_2".modbusMaster.req )
   END_RUNG
   RUNG wire#w1
      { S7_GenerateENO := "TRUE" } Move(in := 1, out1 => "dbTags_master_MPP04_2"."step")
   END_RUNG
   // the same network as SCL:
   // ENO of a box is taken as its EN; it also drops when the box reports an error
   IF ("dbTags_master_MPP04_2"."step" = 12) AND "dbTags_master_MPP04_2".modbusMaster.done THEN
       "dbModbusRTU_Reg".received_6_Stan_urządzenia_1000.typeDataInverter_int[0] := "dbMasterData".data6_Stan_urządzenia_1000.typeDataInverter_int[0];
       "dbTags_master_MPP04_2".modbusMaster.req := FALSE;
       "dbTags_master_MPP04_2"."step" := 1;
   END_IF;
END_REGION

REGION Network 24: Obsługa błędu Modbas / Obsługa błędów Modbaus
   // Obsługa błędu modbus 
   // Inicjacja pętli modbus dla Falownika
   // ustawienie w pętli modbus MPP04-2 krok = 27 ( error modbus)
   // Inicjacja pętli modbus dla następnego urządzenia
   // Ustawienie kroku pętli na stan awaria [27]
   // Uwolnienie linni modbus
   RUNG wire#powerrail
      I_Contact( "FirstScan" )
      { S7_Templates := "SrcType := Word" } NE_Contact(in1 := "dbTags_master_MPP04_2".modbusMaster.errorStatus, in2 := 0)
      Contact( "setErrorModbsmasterMPP04_2" )
      P_Trig( "memRisErrorModbusMPP04_2" )
      wire#w1
      { S7_GenerateENO := "TRUE" } Move(in := 27, out1 => "dbTags_master_MPP04_2"."step")
      { S7_GenerateENO := "TRUE" } Move(in := 0, out1 => "dbModbusRTU_Reg".received_6_Wielkość_przeływu_Adres_0.data[1])
      { S7_GenerateENO := "TRUE" } Move(in := 0, out1 => "dbModbusRTU_Reg".received_6_Wielkość_przeływu_Adres_0.data[0])
   END_RUNG
   RUNG wire#w1
      R_Coil( "dbTags_master_MPP04_2".modbusMaster.req )
   END_RUNG
   // the same network as SCL:
   // ENO of a box is taken as its EN; it also drops when the box reports an error
   #_w1 := NOT "FirstScan" AND ("dbTags_master_MPP04_2".modbusMaster.errorStatus <> 0) AND "setErrorModbsmasterMPP04_2";
   #_w2 := #_w1 AND NOT "memRisErrorModbusMPP04_2";   // rising edge
   "memRisErrorModbusMPP04_2" := #_w1;
   IF #_w2 THEN
       "dbTags_master_MPP04_2"."step" := 27;
       "dbModbusRTU_Reg".received_6_Wielkość_przeływu_Adres_0.data[1] := 0;
       "dbModbusRTU_Reg".received_6_Wielkość_przeływu_Adres_0.data[0] := 0;
       "dbTags_master_MPP04_2".modbusMaster.req := FALSE;
   END_IF;
END_REGION

REGION Network 25: modbus ok / Reset error mdbus status
   // kasowanie statusu błędu
   RUNG wire#powerrail
      { S7_Templates := "SrcType := USInt" } EQ_Contact(in1 := "dbTags_master_MPP04_2"."step", in2 := 12)
      I_Contact( "dbTags_master_MPP04_2".modbusMaster.error )
      wire#w1
      { S7_GenerateENO := "TRUE" } Move(in := 0, out1 => "dbTags_master_MPP04_2".modbusMaster.errorStatus)
   END_RUNG
   RUNG wire#w1
      R_Coil( "dbTags_master_MPP04_2".modbusMaster.done )
   END_RUNG
   // the same network as SCL:
   IF ("dbTags_master_MPP04_2"."step" = 12) AND NOT "dbTags_master_MPP04_2".modbusMaster.error THEN
       "dbTags_master_MPP04_2".modbusMaster.errorStatus := 0;
       "dbTags_master_MPP04_2".modbusMaster.done := FALSE;
   END_IF;
END_REGION

REGION Network 26: Reset Znacznik błedu komunikacji modbus
   RUNG wire#powerrail
      { S7_Templates := "SrcType := USInt" } EQ_Contact(in1 := "dbTags_master_MPP04_2"."step", in2 := 12)
      I_Contact( "dbTags_master_MPP04_2".modbusMaster.error )
      R_Coil( "setErrorModbsmasterMPP04_2" )
   END_RUNG
   // the same network as SCL:
   IF ("dbTags_master_MPP04_2"."step" = 12) AND NOT "dbTags_master_MPP04_2".modbusMaster.error THEN
       "setErrorModbsmasterMPP04_2" := FALSE;
   END_IF;
END_REGION
END_FUNCTION
